// TIA Portal V20 export
FUNCTION_BLOCK "FB - Bas342"   // FB6, LAD
TITLE = Equipment - Bas342
{ S7_Optimized_Access := 'TRUE' }
// This Function blick contain all the logic for controlling a Bas342 module.
// --This module basically for BAS342 sewing machine.
// It is consist of two program bits from BAS342.
// >> Block created by: Engr. Awais Ali
// >> Block creation date:  08-10-2025
// stored: MemoryReserve 100, SetENOAutomatically false
   VAR_INPUT
      i_xProgrambit0 : Bool;
      i_xProgrambit1 : Bool;
   END_VAR
   VAR_IN_OUT
      iq_Bas342 : "UDT-BAS342";
   END_VAR
BEGIN

REGION Network 1: Control - left jig
   // Bit 0 represent the left jig program.
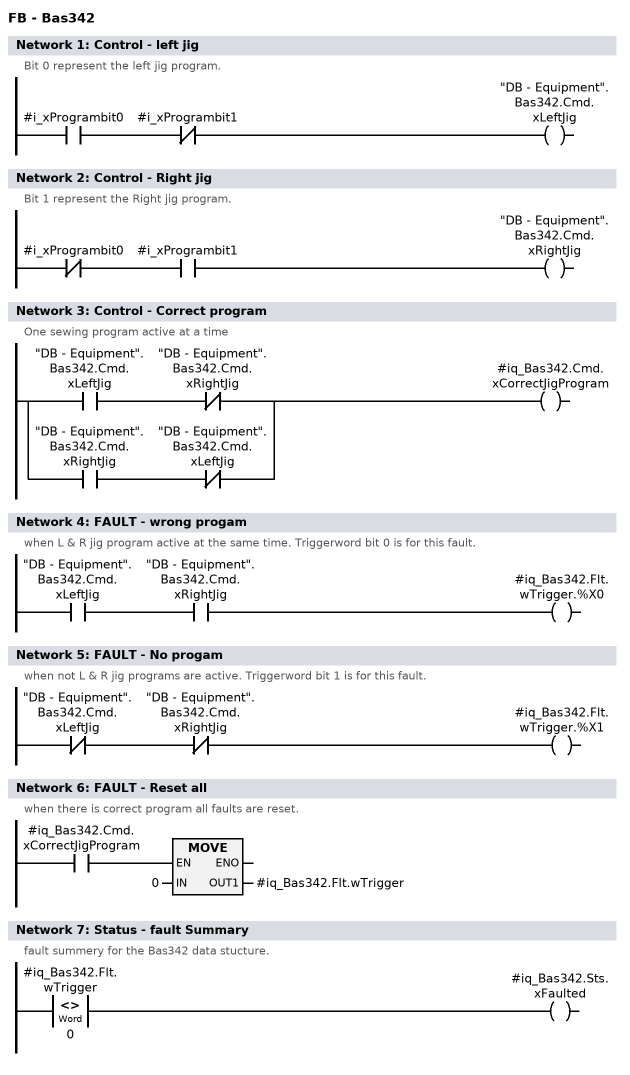
   RUNG wire#powerrail
      Contact( #i_xProgrambit0 )
      I_Contact( #i_xProgrambit1 )
      Coil( "DB - Equipment".Bas342.Cmd.xLeftJig )
   END_RUNG
   // the same network as SCL:
   "DB - Equipment".Bas342.Cmd.xLeftJig := #i_xProgrambit0 AND NOT #i_xProgrambit1;
END_REGION

REGION Network 2: Control - Right jig
   // Bit 1 represent the Right jig program.
   RUNG wire#powerrail
      I_Contact( #i_xProgrambit0 )
      Contact( #i_xProgrambit1 )
      Coil( "DB - Equipment".Bas342.Cmd.xRightJig )
   END_RUNG
   // the same network as SCL:
   "DB - Equipment".Bas342.Cmd.xRightJig := NOT #i_xProgrambit0 AND #i_xProgrambit1;
END_REGION

REGION Network 3: Control - Correct program
   // One sewing program active at a time
   RUNG wire#powerrail
      Contact( "DB - Equipment".Bas342.Cmd.xLeftJig )
      I_Contact( "DB - Equipment".Bas342.Cmd.xRightJig )
      wire#w1
      Coil( #iq_Bas342.Cmd.xCorrectJigProgram )
   END_RUNG
   RUNG wire#powerrail
      Contact( "DB - Equipment".Bas342.Cmd.xRightJig )
      I_Contact( "DB - Equipment".Bas342.Cmd.xLeftJig )
   END_RUNG wire#w1
   // the same network as SCL:
   #iq_Bas342.Cmd.xCorrectJigProgram := ("DB - Equipment".Bas342.Cmd.xLeftJig AND NOT "DB - Equipment".Bas342.Cmd.xRightJig) OR ("DB - Equipment".Bas342.Cmd.xRightJig AND NOT "DB - Equipment".Bas342.Cmd.xLeftJig);
END_REGION

REGION Network 4: FAULT - wrong progam
   // when L & R jig program active at the same time. Triggerword bit 0 is for this fault.
   RUNG wire#powerrail
      Contact( "DB - Equipment".Bas342.Cmd.xLeftJig )
      Contact( "DB - Equipment".Bas342.Cmd.xRightJig )
      Coil( #iq_Bas342.Flt.wTrigger.%X0 )
   END_RUNG
   // the same network as SCL:
   #iq_Bas342.Flt.wTrigger.%X0 := "DB - Equipment".Bas342.Cmd.xLeftJig AND "DB - Equipment".Bas342.Cmd.xRightJig;
END_REGION

REGION Network 5: FAULT - No progam
   // when not L & R jig programs are active. Triggerword bit 1 is for this fault.
   RUNG wire#powerrail
      I_Contact( "DB - Equipment".Bas342.Cmd.xLeftJig )
      I_Contact( "DB - Equipment".Bas342.Cmd.xRightJig )
      Coil( #iq_Bas342.Flt.wTrigger.%X1 )
   END_RUNG
   // the same network as SCL:
   #iq_Bas342.Flt.wTrigger.%X1 := NOT "DB - Equipment".Bas342.Cmd.xLeftJig AND NOT "DB - Equipment".Bas342.Cmd.xRightJig;
END_REGION

REGION Network 6: FAULT - Reset all
   // when there is correct program all faults are reset.
   RUNG wire#powerrail
      Contact( #iq_Bas342.Cmd.xCorrectJigProgram )
      Move(in := 0, out1 => #iq_Bas342.Flt.wTrigger)
   END_RUNG
   // the same network as SCL:
   IF #iq_Bas342.Cmd.xCorrectJigProgram THEN #iq_Bas342.Flt.wTrigger := 0; END_IF;
END_REGION

REGION Network 7: Status - fault Summary
   // fault summery for the Bas342 data stucture.
   RUNG wire#powerrail
      { S7_Templates := "SrcType := Word" } NE_Contact(in1 := #iq_Bas342.Flt.wTrigger, in2 := 0)
      Coil( #iq_Bas342.Sts.xFaulted )
   END_RUNG
   // the same network as SCL:
   #iq_Bas342.Sts.xFaulted := #iq_Bas342.Flt.wTrigger <> 0;
END_REGION
END_FUNCTION_BLOCK
